// Mitsubishi GX Works2 project: 시뭔스 무한반복 예제2 (수제)   PLC: Q03UDV

PROGRAM MAIN
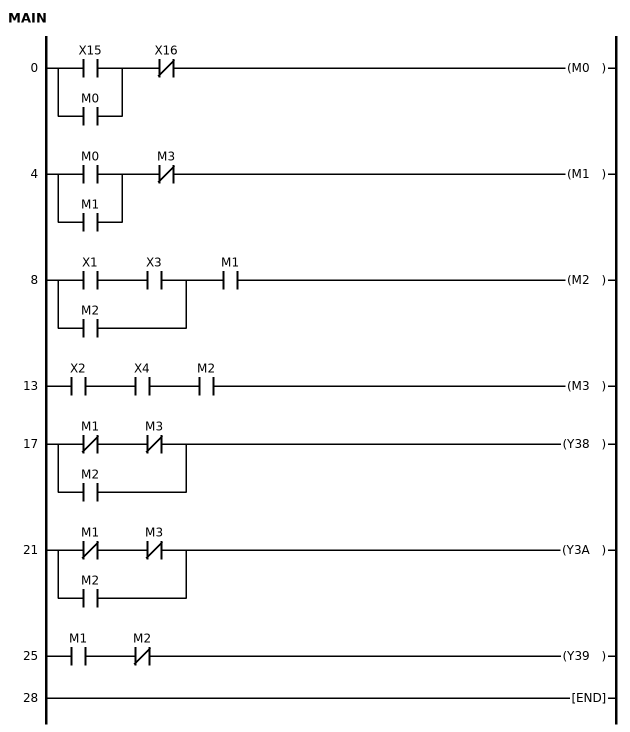
0     LD      X15
      OR      M0
      ANI     X16
      OUT     M0
4     LD      M0
      OR      M1
      ANI     M3
      OUT     M1
8     LD      X1
      AND     X3
      OR      M2
      AND     M1
      OUT     M2
13    LD      X2
      AND     X4
      AND     M2
      OUT     M3
17    LDI     M1
      ANI     M3
      OR      M2
      OUT     Y38
21    LDI     M1
      ANI     M3
      OR      M2
      OUT     Y3A
25    LD      M1
      ANI     M2
      OUT     Y39
28    END
END_PROGRAM
